FUNCTION_BLOCK Insertion2D
VAR_INPUT
	slider : I_LinearEncodedDrive;
	screw : I_LinearContinuousDrive;
END_VAR
VAR_OUTPUT
	contact AT %I* : BOOL;
	
	active : BOOL;
	error : BOOL;
	home : BOOL;
	
	homingComplete : BOOL;
	
	sliderPos : LREAL;
END_VAR
(*
this FB encapsulates 2 linear drives (1 encoded slider, 1 continuous screw) into a generic insertion machine
both drives should be declared and called externally as a concrete FB
*)

homingComplete := slider.HomeSet AND screw.HomeSet;

active := slider.Active OR screw.Active;
error := slider.Error OR screw.Error;
home := slider.AtHome AND screw.AtHome;

sliderPos := slider.CurrentPosition;

METHOD align : BOOL
VAR_INPUT
	targetPos : REAL;
END_VAR
{warning disable C0371}
slider.moveAbsolute(newTarget := targetPos);
END_METHOD

METHOD homingSequence : BOOL
VAR_INPUT
END_VAR
{warning disable C0371}
IF NOT slider.homeSet THEN
	slider.homingSequence();
END_IF

IF NOT screw.homeSet THEN
	screw.homingSequence();
END_IF

homingSequence := homingComplete;
END_METHOD

METHOD press : BOOL
VAR_INPUT
END_VAR
{warning disable C0371}
IF NOT contact THEN
	screw.moveContinuous(newDirection := MC_Negative_Direction);
END_IF
END_METHOD

METHOD release : BOOL
VAR_INPUT
END_VAR
{warning disable C0371}
screw.moveContinuous(newDirection := MC_Positive_Direction);
END_METHOD

METHOD reset : BOOL
VAR_INPUT
END_VAR
{warning disable C0371}
slider.reset();
screw.reset();
END_METHOD

METHOD stop : BOOL
VAR_INPUT
END_VAR
{warning disable C0371}
screw.stop();
slider.stop();
END_METHOD

METHOD toHome : BOOL
VAR_INPUT
END_VAR
{warning disable C0371}
slider.toHome();
screw.toHome();

toHome := slider.AtHome AND screw.AtHome;
END_METHOD

METHOD traverse : BOOL
VAR_INPUT
	direction : MC_Direction;
END_VAR
{warning disable C0371}
slider.moveContinuous(newDirection:= direction);
END_METHOD

END_FUNCTION_BLOCK

(* stored: Version 1.1.0.1, ProductVersion 3.1.4024.11
   POU Insertion2D: Id {fd3338dd-9255-4680-9ae4-db8063fef1d5}, SpecialFunc None
   Method align: Id {47a93987-1e63-457b-976d-e3beb6a85a58}
   Method homingSequence: Id {a490d2f3-e9c5-442b-9291-a1ccc0f2ac16}
   Method press: Id {a04032fe-cf9f-475c-8ef3-620016e2c35d}
   Method release: Id {4fcd5174-6951-4a0e-a154-3a5ff87fdd59}
   Method reset: Id {2a5e1a57-ae80-40dc-b7af-1829d7712c98}
   Method stop: Id {880cadeb-51df-4dbe-b47b-f6f226727247}
   Method toHome: Id {0588376b-b19c-46ad-8507-63727c94039a}
   Method traverse: Id {1776946c-feed-460c-83a0-f2c05c981663} *)
